(*********************************** G.D S.p.A. - Technical Department ***********************************
============= PROGRAM INFO ============
FOLDER:             TBD
MACHINES INVOLVED:  TBD 

============= DESCRIPTION =============
csp machine declaration

============= REVISIONS ===============
Date		Version	 	Author      	Description             
----------	-------		------------  	--------------------------------------------
2019/04/05 	0000.00	 	M.Grasso		Creation of the PRG

**********************************************************************************************************)
(*$R process_ref := prc; $*)
PROGRAM csp_case_tr_squaring_os
VAR
	
	prc:											process;
	prc_path:										STRING;
	
END_VAR

_read_var_input();

_object_manager();

IF NOT objects_running()
THEN
	RETURN;	
END_IF

_read_process_image();

_mode_manager();

_set_runtime_properties();

(********************************* BODY *********************************)
(************************************************************************)

_handle_messages();

_write_output();

ACTION _handle_messages:
;
END_ACTION

ACTION _handle_process_test:
;
END_ACTION

ACTION _mode_manager:
IF process_mode_req_is_pending(prc)
THEN
    process_apply_mode_req_first_step(prc);
    CASE process_get_mode(prc) OF
        MODE_TO_ABSENT:
			;
        MODE_TO_INACTIVE:
			;
        MODE_TO_TEST:
			;
        MODE_TO_OPERATIONAL:
			;
    END_CASE
    process_apply_mode_req_second_step(prc);
END_IF
END_ACTION

ACTION _object_manager:
IF objects_initialization()
THEN
	sub_process_init(
		object_name					:= 'csp_case_tr_squaring_os.prc', 
		process						:= csp_case_topRail_squaring.prc, 
		CONVERSION_this				:= prc);
		
	prc_path 						:= process_get_path(prc);
END_IF

IF objects_running()
THEN
	process_cycle(prc);
END_IF
END_ACTION

ACTION _read_process_image:
;
END_ACTION

ACTION _read_var_input:
;
END_ACTION

ACTION _set_runtime_properties:
;
END_ACTION

ACTION _write_output:
;
END_ACTION

END_PROGRAM

(* stored: Version 1.1.0.1, ProductVersion 3.1.4022.12
   POU csp_case_tr_squaring_os: Id {b7295895-8343-4f3e-ac3a-3d8f931ac93b}, SpecialFunc None
   Action _handle_messages: Id {777cfee9-a104-48a9-a9c6-81f4b0eec376}
   Action _handle_process_test: Id {9f9a6984-4ed0-46c7-8c6b-c6e4f67c151b}
   Action _mode_manager: Id {f6156f74-729b-4b9c-9569-46002b2e1aa9}
   Action _object_manager: Id {5e75b884-c28d-42cc-a9a6-7b337583d1c3}
   Action _read_process_image: Id {870b63ba-cefe-4eed-a977-012c7298c9e9}
   Action _read_var_input: Id {8d042e83-1cbf-47f5-9e47-9875e5a66c06}
   Action _set_runtime_properties: Id {1a09b145-05c3-4156-ae9a-4384aaf06be9}
   Action _write_output: Id {5e6ce9ba-1fa6-44d9-a0e2-45ede3222871} *)
